PROGRAM NEWSUBROUTINE

VAR_INPUT
	input	:BOOL;	
END_VAR
VAR
	c1		:CTD;
	counter2 :LREAL:=3.5;
	
END_VAR

//c1(
//	CD:= , 
//	LOAD:= , 
//	PV:= , 
//	Q=> , 
//	CV=> );


//IF input = TRUE THEN
//	counter2 := counter2 + 1;
//ELSE
//	counter2 := counter2 - 1;
//END_IF

END_PROGRAM

(* stored: Version 1.1.0.1, ProductVersion 3.1.4024.13
   POU NEWSUBROUTINE: Id {1dfba1ce-1774-4278-82cf-8990bce4e998}, SpecialFunc None *)
